// TIA Portal V19 export
VAR_GLOBAL   // PLC tag table "D01"
   D01_Lp_EntryReq_LB101 AT %Q106.3 : Bool;   // 188SH1
   D01_Lp_SafetyReset_LB101 AT %Q106.4 : Bool;   // 188SH2
   D01_Pb_EntryReq_LB101 AT %I102.7 : Bool;   // 188SH1
   D01_Pb_SafetyReset_LB101 AT %I103.0 : Bool;   // 188SH2
   D01_Ls AT %I1020.0 : Bool;   // 102DI0 - 188BE1/R1
END_VAR
